PROGRAM MQ_FSY
VAR
//	CS_FSY_TcpAn: CS_FsyTcp;
	CS_FSY_TcpCa: CS_FsyTcp;
	Cold_step :UINT;
	scan_TON1 :Tc2_Standard.TON;
	Scan_TON :ARRAY[1..7] OF Tc2_Standard.TON;
	Scan_code_Z : R_TRIG;
	I:INT;
END_VAR

//扫码



Saoma();
P3User2_Par.MQ_AnFSY_IP:='192.168.10.40';
P3User2_Par.MQ_CaFSY_IP:='192.168.10.41';
Scan_TON[1](PT:=T#1MS);
Scan_TON[2](PT:=T#1MS);
Scan_TON[3](PT:=T#1MS);
Scan_TON[4](PT:=T#100MS);

Scan_code_Z (CLK:=Cold_Scan_code, Q=>);

IF Scan_code_Z.Q AND  Cold_step=0 THEN
	 Cold_step:=10;
END_IF




CASE Cold_step OF
0:
	IF Scan_start AND NOT bCodeError AND NOT bCodeConError AND NOT P3User2_Par.Shield[4] THEN
	 Cold_step:=10;
	 Code_State:=0;
	ELSIF P3User2_Par.Shield[4] THEN
	 Cold_step:=70;
	END_IF
10:
	Scan_TON[1].IN:=FALSE;
	Scan_TON[2].IN:=FALSE;
	Scan_TON[3].IN:=FALSE;
	Cold_step:=20;
	
20:
	bScan_init:=TRUE;
	Scan_TON[1].IN:=TRUE;
	IF Scan_TON[1].Q THEN
		bScan_init:=FALSE;
		Scan_TON[1].IN:=FALSE;
		Cold_step:=30;
	END_IF

30:
	bTcpOpen:=TRUE;
	Scan_TON[2].IN:=TRUE;
	IF Scan_TON[2].Q THEN
		bTcpOpen:=FALSE;
		Scan_TON[2].IN:=FALSE;
		Cold_step:=40;
	END_IF

40:
	IF bTcpOpen_OK THEN
		Cold_step:=50;
	END_IF

50:
	bScan_start:=TRUE;
	Scan_TON[3].IN:=TRUE;
	IF Scan_TON[3].Q THEN
		bScan_start:=FALSE;
		Scan_TON[3].IN:=FALSE;
		Cold_step:=60;
	END_IF
60:
	Scan_TON[4].IN:=TRUE;
	IF 	Scan_TON[4].Q THEN
		Cold_step:=70;
		Scan_TON[4].IN:=FALSE;
	END_IF

70:
IF NOT P3User2_Par.Shield[4] THEN
	IF Code_State=1 AND (strCode<>'') THEN
		CellMemory[CellNo.OvenMoveClip1].Cell_number1:=strCode;
		IF strCode=CellMemory[CellNo.OvenMoveClip1].Cell_number THEN
			CellMemory[CellNo.OvenMoveClip1].ScanCode:=1;
			Scan_start:=FALSE;
			Scan_finish:=TRUE;
			Cold_step:=80;				
			I:=0;
		ELSIF strCode<>CellMemory[CellNo.OvenMoveClip1].Cell_number THEN
			CellMemory[CellNo.OvenMoveClip1].ScanCode:=2;
			P3_Error[79]:=TRUE;//冷压扫码第二次扫码校验NG
			Scan_start:=FALSE;
			Scan_finish:=TRUE;
			Cold_step:=80;
			I:=0;
		END_IF
	ELSIF  Code_State=2 AND I<3 THEN
			Cold_step:=10;
			I:=I+1;		
	ELSIF Code_State=2 AND I>=3 THEN
		CellMemory[CellNo.ColdpressClip].Cell_number1:=strCode;
		CellMemory[CellNo.ColdpressClip].ScanCode:=2;
		P3_Error[16]:=TRUE;//冷压扫码NG报警
		Scan_start:=FALSE;
		Scan_finish:=TRUE;
		Cold_step:=80;
		I:=0;
	END_IF
ELSIF P3User2_Par.Shield[4] THEN
		CellMemory[CellNo.OvenMoveClip1].Cell_number1:='A1234567890ABCDEF';
		CellMemory[CellNo.OvenMoveClip1].ScanCode:=1;
		Scan_start:=FALSE;
		Scan_finish:=TRUE;
		Cold_step:=80;				
		I:=0;
END_IF
80:
	IF NOT Scan_finish THEN
		Cold_step:=0;
	END_IF
END_CASE

ACTION Saoma:
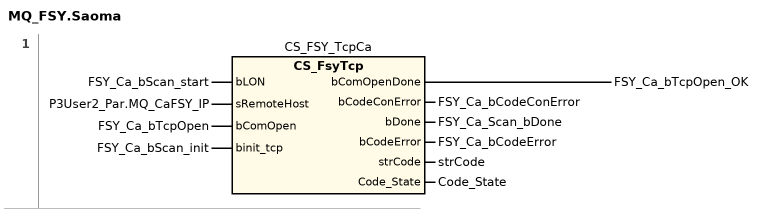
// NETWORK 1
CS_FSY_TcpCa(
    bLON := FSY_Ca_bScan_start,
    sRemoteHost := P3User2_Par.MQ_CaFSY_IP,
    bComOpen := FSY_Ca_bTcpOpen,
    binit_tcp := FSY_Ca_bScan_init,
    bCodeConError => FSY_Ca_bCodeConError,
    bDone => FSY_Ca_Scan_bDone,
    bCodeError => FSY_Ca_bCodeError,
    strCode => strCode,
    Code_State => Code_State); // CS_FsyTcp
FSY_Ca_bTcpOpen_OK := CS_FSY_TcpCa.bComOpenDone;
END_ACTION

END_PROGRAM

(* stored: Version 1.1.0.1, ProductVersion 3.1.4024.12
   POU MQ_FSY: Id {f97cd1b8-59c0-43fd-b436-c814d3cb837d}, SpecialFunc None
   Action Saoma: Id {b4e57f1d-587e-4fee-afee-22bfaecb448b} *)
